Omron CX-Programmer project NewProject (CX-Programmer 9.75)

# PLC omron: CP1E N30

## Global symbols (name address type ; comment)
T000 BOOL  ; T0
T001 BOOL  ; T01
T002 BOOL  ; T02
T003 BOOL  ; T03
T004 BOOL  ; T04
T005 BOOL  ; T05

## Program NewProgram1 (cyclic task 0)
Local symbols
cm1 100.04 BOOL
cpm 100.06 BOOL
lm 100.07 BOOL
mps 100.00 BOOL
sensor 0.03 BOOL
sensor1 0.05 BOOL
start 0.00 BOOL
stop 0.01 BOOL
v1 100.04 BOOL

### Section Section1

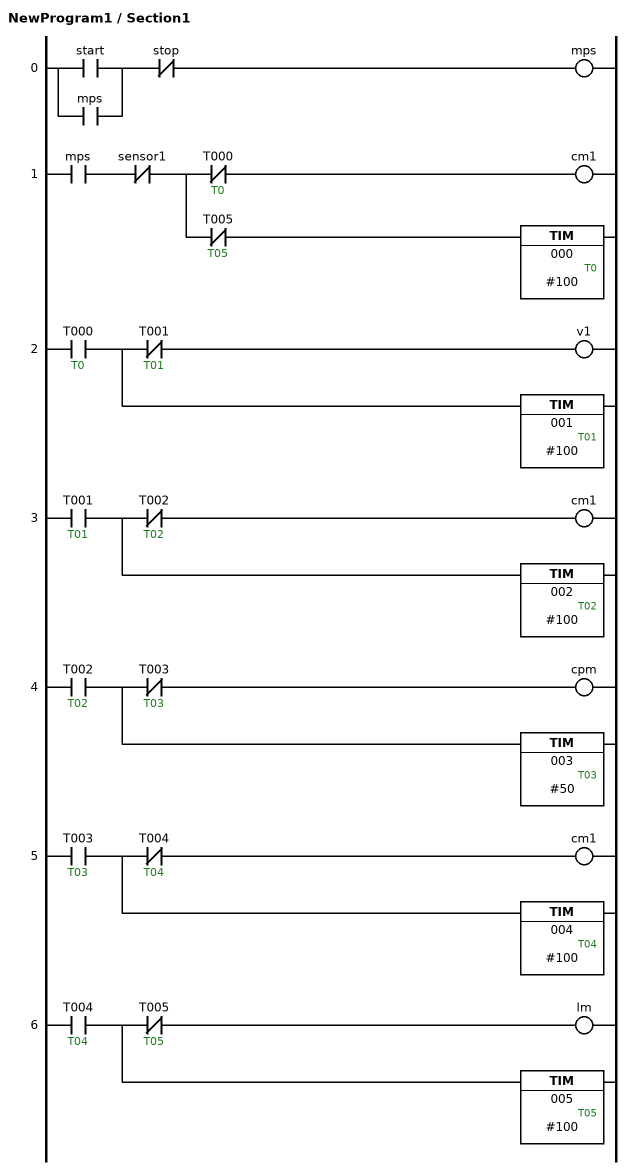
; rung 0
LD start
OR mps
ANDNOT stop
OUT mps
; rung 1
LD mps
ANDNOT sensor1
OUT TR0
ANDNOT T000  ; T0
OUT cm1
LD TR0
ANDNOT T005  ; T05
TIM 000 #100  ; T0
; rung 2
LD T000  ; T0
OUT TR0
ANDNOT T001  ; T01
OUT v1
LD TR0
TIM 001 #100  ; T01
; rung 3
LD T001  ; T01
OUT TR0
ANDNOT T002  ; T02
OUT cm1
LD TR0
TIM 002 #100  ; T02
; rung 4
LD T002  ; T02
OUT TR0
ANDNOT T003  ; T03
OUT cpm
LD TR0
TIM 003 #50  ; T03
; rung 5
LD T003  ; T03
OUT TR0
ANDNOT T004  ; T04
OUT cm1
LD TR0
TIM 004 #100  ; T04
; rung 6
LD T004  ; T04
OUT TR0
ANDNOT T005  ; T05
OUT lm
LD TR0
TIM 005 #100  ; T05

### Section END
; rung 0
END(001)